PROGRAM MainControl
VAR
	fbErrorHandling : FB_ErrorHandling;
	fbServiceModule : FB_ServiceModule;
	fbLevitationSystem : FB_LevitationSystem;
	fbGuidanceSystem : FB_GuidanceSystem;
	
	stFromOperationControlToMainControl : FromOperationControlToMainControl;
	stFromMainControlToOperationControl : FromMainControlToOperationControl;
	
	eMainState : eMainStateMachine := eMainStateMachine.STARTUP;
	
	fbErrorTimer : TON := (PT := T#10S);
	bStartUpError : BOOL;
	bGoToError : BOOL;
	
	bOnGround : BOOL;

	
	nMode : BYTE := 0;
	
END_VAR

fbErrorHandling();

CASE eMainState OF
	//
	eMainStateMachine.STARTUP:
		doEnableSubsystems();
		doCallSubsystems();
		doCheckSystem();
	//
	eMainStateMachine.READY:
		doCallSubsystems();
		doActivateHighLevelSTM();
		
		IF fbErrorHandling.getGoToERROR THEN
			fbServiceModule.eState := eServiceModuleSTM.PreparingForError;
		ELSE
			fbServiceModule.eState := eServiceModuleSTM.Waiting;
		END_IF

	
		IF fbErrorHandling.getGoToERROR THEN
			eMainState := eMainStateMachine.ERROR;
		ELSIF stFromOperationControlToMainControl.OM_origO_StartOperational THEN
			eMainState := eMainStateMachine.OPERATIONAL;
		END_IF

	//
	eMainStateMachine.OPERATIONAL:
		doCallSubsystems();
		
		fbServiceModule.eState := eServiceModuleSTM.Running;
		
		
		IF fbErrorHandling.getGoToSHUTDOWN OR stFromOperationControlToMainControl.OM_origO_StopOperational THEN
			eMainState := eMainStateMachine.SHUTDOWN;
		ELSE
			eMainState := eMainStateMachine.OPERATIONAL;
		END_IF
	//
	eMainStatemachine.SHUTDOWN:
		doCallSubsystems();
		
		IF fbErrorHandling.getGoToSHUTDOWN THEN
			fbServiceModule.eState := eServiceModuleSTM.PreparingForError;
		ELSE
			fbServiceModule.eState := eServiceModuleSTM.PostRunning;
		END_IF
		
		
		
		IF bOnGround THEN
			IF fbErrorHandling.getGoToSHUTDOWN THEN
				eMainState := eMainStateMachine.ERROR;
			ELSE
				eMainState := eMainStateMachine.READY;
			END_IF
		END_IF
	//	
	eMainStateMachine.ERROR:
		
		IF stFromOperationControlToMainControl.OM_origO_AckError THEN
			eMainState := eMainStateMachine.STARTUP;
		END_IF

END_CASE

METHOD PRIVATE doActivateHighLevelSTM
VAR_INPUT
END_VAR
CASE nMode OF
	0:	fbServiceModule.bSTMActive := TRUE;
		fbLevitationSystem.setActive := TRUE;
		fbGuidanceSystem.setActive := TRUE;
	
	1:	fbLevitationSystem.setActive := TRUE;
		fbGuidanceSystem.setActive := TRUE;
	
	2:	fbServiceModule.bSTMActive := TRUE;
		fbGuidanceSystem.setActive := TRUE;
	
	4:	fbServiceModule.bSTMActive := TRUE;
		fbLevitationSystem.setActive := TRUE;
	
	3:	fbGuidanceSystem.setActive := TRUE;
	
	5:	fbLevitationSystem.setActive := TRUE;
	
	6:	fbServiceModule.bSTMActive := TRUE;
END_CASE
END_METHOD

METHOD doCallSubsystems
VAR_INPUT
END_VAR
CASE nMode OF
	0:
		fbServiceModule();
		fbLevitationSystem();
		fbGuidanceSystem();
	1:
		fbLevitationSystem();
		fbGuidanceSystem();
	2:
		fbServiceModule();
		fbGuidanceSystem();
	4:
		fbServiceModule();
		fbLevitationSystem();
	3:
		fbGuidanceSystem();
	5:
		fbLevitationSystem();
	6:
		fbServiceModule();
END_CASE
END_METHOD

METHOD doCheckSystem
VAR_INPUT
END_VAR
VAR	
END_VAR
CASE nMode OF
	0:	//All Enabled
		IF fbServiceModule.eCondition = eConditionCheck.RUN AND fbLevitationSystem.eCondition = eConditionCheck.RUN AND fbGuidanceSystem.eCondition = eConditionCheck.RUN THEN
			fbErrorTimer(IN := FALSE);
			eMainState := eMainStateMachine.READY;
		ELSE
			fbErrorTimer(IN := TRUE);
			IF fbErrorTimer.Q THEN
				bStartUpError := TRUE;
				fbErrorTimer(IN := FALSE);
				eMainState := eMainStateMachine.ERROR;
			ELSE
				eMainState := eMainStateMachine.STARTUP;
			END_IF
		END_IF
		
	1:	//ServiceModule Disabled
		IF fbLevitationSystem.eCondition = eConditionCheck.RUN AND fbGuidanceSystem.eCondition = eConditionCheck.RUN THEN
			fbErrorTimer(IN := FALSE);
			
			eMainState := eMainStateMachine.READY;
		ELSE
			fbErrorTimer(IN := TRUE);
			IF fbErrorTimer.Q THEN
				bStartUpError := TRUE;
				fbErrorTimer(IN := FALSE);
				eMainState := eMainStateMachine.ERROR;
			ELSE
				eMainState := eMainStateMachine.STARTUP;
			END_IF
		END_IF
		
	2: //Levitation Disabled
		IF fbServiceModule.eCondition = eConditionCheck.RUN AND fbGuidanceSystem.eCondition = eConditionCheck.RUN THEN
			fbErrorTimer(IN := FALSE);
			eMainState := eMainStateMachine.READY;
		ELSE
			fbErrorTimer(IN := TRUE);
			IF fbErrorTimer.Q THEN
				bStartUpError := TRUE;
				fbErrorTimer(IN := FALSE);
				eMainState := eMainStateMachine.ERROR;
			ELSE
				eMainState := eMainStateMachine.STARTUP;
			END_IF
		END_IF

	4: //Guidance Disabled	
		IF fbServiceModule.eCondition = eConditionCheck.RUN AND fbLevitationSystem.eCondition = eConditionCheck.RUN THEN
			fbErrorTimer(IN := FALSE);
			eMainState := eMainStateMachine.READY;
		ELSE
			fbErrorTimer(IN := TRUE);
			IF fbErrorTimer.Q THEN
				bStartUpError := TRUE;
				fbErrorTimer(IN := FALSE);
				eMainState := eMainStateMachine.ERROR;
			ELSE
				eMainState := eMainStateMachine.STARTUP;
			END_IF
		END_IF
		
	3: //ServiceModule and Levitation Disabled
		IF fbGuidanceSystem.eCondition = eConditionCheck.RUN THEN
			fbErrorTimer(IN := FALSE);
			eMainState := eMainStateMachine.READY;
		ELSE
			fbErrorTimer(IN := TRUE);
			IF fbErrorTimer.Q THEN
				bStartUpError := TRUE;
				fbErrorTimer(IN := FALSE);
				eMainState := eMainStateMachine.ERROR;
			ELSE
				eMainState := eMainStateMachine.STARTUP;
			END_IF
		END_IF
		
	5: //ServiceModule and Guidance Disabled
		IF fbLevitationSystem.eCondition = eConditionCheck.RUN THEN
			fbErrorTimer(IN := FALSE);
			eMainState := eMainStateMachine.READY;
		ELSE
			fbErrorTimer(IN := TRUE);
			IF fbErrorTimer.Q THEN
				bStartUpError := TRUE;
				fbErrorTimer(IN := FALSE);
				eMainState := eMainStateMachine.ERROR;
			ELSE
				eMainState := eMainStateMachine.STARTUP;
			END_IF
		END_IF
		
	6: //Levitation and Guidance Disabled
		IF fbServiceModule.eCondition = eConditionCheck.RUN THEN
			fbErrorTimer(IN := FALSE);
			eMainState := eMainStateMachine.READY;
		ELSE
			fbErrorTimer(IN := TRUE);
			IF fbErrorTimer.Q THEN
				bStartUpError := TRUE;
				fbErrorTimer(IN := FALSE);
				eMainState := eMainStateMachine.ERROR;
			ELSE
				eMainState := eMainStateMachine.STARTUP;
			END_IF
		END_IF
		
	7: //All Disabled
		fbErrorTimer(IN := TRUE);
		IF fbErrorTimer.Q THEN
			bStartUpError := TRUE;
			fbErrorTimer(IN := FALSE);
			eMainState := eMainStateMachine.ERROR;
		ELSE
			eMainState := eMainStateMachine.STARTUP;
		END_IF
END_CASE
END_METHOD

METHOD PRIVATE doDataHandling
VAR_INPUT
END_VAR
END_METHOD

METHOD doEnableSubsystems
VAR_INPUT
END_VAR
nMode.0 := stFromOperationControlToMainControl.OM_origO_ServiceModuleDisabled;
nMode.1 := stFromOperationControlToMainControl.OM_origO_LevitationDisable;
nMode.2 := stFromOperationControlToMainControl.OM_origO_GuidanceDisable;
END_METHOD

END_PROGRAM

(* stored: Version 1.1.0.1, ProductVersion 3.1.4024.12
   POU MainControl: Id {165fa4b6-fe79-4748-9022-b33b5b722466}, SpecialFunc None
   Method doActivateHighLevelSTM: Id {47446e0a-b75b-4c67-8d8c-35029d1ee551}
   Method doCallSubsystems: Id {c330acab-a3df-4219-8ed4-48f648a160a3}
   Method doCheckSystem: Id {55b5a3ff-6d8a-4578-a9a0-1bbfe6d7f606}
   Method doDataHandling: Id {6650b2a5-53d2-4d59-90c1-16aa8c80f746}
   Method doEnableSubsystems: Id {4402bbf9-07a3-41dd-916a-44a19b1d489b} *)
